(* PLC project TestPLC, Beckhoff Automation GmbH TwinCAT PLC Control 3.5.8.40 *)
(* stored: creationDateTime 2017-11-15T09:25:53.0336397, modificationDateTime 2017-11-15T09:25:53.0336397 *)

PROGRAM MAIN
VAR 
	iTest:INT;
	bTest:BOOL;
	iTest2:INT;
	
	tobias:BOOL;
	
END_VAR

            iTest:=iTest+1;

IF iTest2<0
	THEN iTest2:=1;
	ELSE iTest2:=iTest2+100;
END_IF

tobias:=TRUE;


          
END_PROGRAM
